// TwinCAT 3 PLC project PLCStudent
// ProgramVersion: 3.1.4022.3
// libraries:
//   Tc2_Standard, * (Beckhoff Automation GmbH)
//   Tc2_System, * (Beckhoff Automation GmbH)
//   Tc3_Module, * (Beckhoff Automation GmbH)
// project tree:
//   GVLs/ GVL.TcGVL
//   / PlcTask.TcTTO (not stored)
//   POUs/ MAIN.TcPOU, Wash.TcPOU
// (motion and I/O tree: see PLC project plcsim)
// real-time tasks:
//   TASK PlcTask: cycle T#80ms, priority 1, ADS port 350
//   TASK PlcTask1: cycle T#10ms, priority 20, ADS port 351
// variable links:
//   PLCSim/PLCSim Instance <-> PLCStudent/PLCStudent Instance
//     PlcTask Inputs/GVL.ixBack <-> PlcTask Outputs/GVL.qxBack
//     PlcTask Inputs/GVL.ixDispBit1 <-> PlcTask Outputs/GVL.qxDispBit1
//     PlcTask Inputs/GVL.ixDispBit2 <-> PlcTask Outputs/GVL.qxDispBit2
//     PlcTask Inputs/GVL.ixDrain <-> PlcTask Outputs/GVL.qxDrain
//     PlcTask Inputs/GVL.ixFill <-> PlcTask Outputs/GVL.qxFill
//     PlcTask Inputs/GVL.ixForw <-> PlcTask Outputs/GVL.qxForw
//     PlcTask Inputs/GVL.ixHeating <-> PlcTask Outputs/GVL.qxHeatingON
//     PlcTask Inputs/GVL.ixPulseTwo <-> PlcTask Outputs/GVL.qxPulseTwo
//     PlcTask Inputs/GVL.ixSpin <-> PlcTask Outputs/GVL.qxSpin
//     PlcTask Outputs/GVL.qwCurTemp <-> PlcTask Inputs/GVL.iwCurrentTemp
//     PlcTask Outputs/GVL.qwSetTem <-> PlcTask Inputs/GVL.iwSetTemp
//     PlcTask Outputs/GVL.qxLevel1 <-> PlcTask Inputs/GVL.ixLevel1
//     PlcTask Outputs/GVL.qxLevel2 <-> PlcTask Inputs/GVL.ixLevel2
//     PlcTask Outputs/GVL.qxLevel3 <-> PlcTask Inputs/GVL.ixLevel3
//     PlcTask Outputs/GVL.qxNotEmpty <-> PlcTask Inputs/GVL.ixNotEmpty
//     PlcTask Outputs/GVL.qxPulseOne <-> PlcTask Inputs/GVL.ixPulseOne
//     PlcTask Outputs/GVL.qxSetLevel <-> PlcTask Inputs/GVL.ixSetLevel
//     PlcTask Outputs/GVL.qxStart <-> PlcTask Inputs/GVL.ixStart
//     PlcTask Outputs/GVL.qxTempOk <-> PlcTask Inputs/GVL.ixTempOk

// ---- GVLs/GVL.TcGVL
{attribute 'qualified_only'}
VAR_GLOBAL
	ixPulseOne		AT %I*:	BOOL; 		(* PULS button *)
	ixStart			AT %I*:	BOOL; 		(* START switch *)
	ixSetLevel		AT %I*:	BOOL; 		(* NIVÅ switch *)
	ixLevel3		AT %I*:	BOOL; 		(* Sensor for level 3 *)
	ixLevel2		AT %I*:	BOOL; 		(* Sensor for level 2 *)
	ixLevel1		AT %I*:	BOOL; 		(* Sensor for level 1 *)
	ixNotEmpty		AT %I*:	BOOL; 		(* Sensor for not empty *)
	ixTempOk		AT %I*:	BOOL; 		(* Temp sensor *)
	iwSetTemp		AT %I*: INT;		(* Temparature set on the dail in HMI*)
	iwCurrentTemp	AT %I*: INT;		(* Current Temparture of the washing machine*)
	
	qxPulseTwo		AT %Q*:	BOOL; 		(* PULS button *)
	qxForw			AT %Q*:	BOOL; 		(* Washer cylinder forward *)
	qxBack			AT %Q*:	BOOL; 		(* Washer cylinder back *)
	qxSpin			AT %Q*:	BOOL; 		(* Washer cylinder spin *)
	qxFill			AT %Q*:	BOOL; 		(* Fill water *)
	qxDrain			AT %Q*:	BOOL; 		(* Drain water *)
	qxDispBit1		AT %Q*:	BOOL; 		(* Display bit 1 *)
	qxDispBit2		AT %Q*:	BOOL; 		(* Display bit 2 *)
	qxHeatingON		AT %Q*: BOOL;		(* Heater ON *)
END_VAR

// ---- POUs/MAIN.TcPOU
PROGRAM MAIN
VAR
END_VAR

Wash();

END_PROGRAM

// ---- POUs/Wash.TcPOU
PROGRAM Wash
VAR
	Blink_Timer: TP;
	Stop_Timer: TON;
	Memorize: BOOL;
END_VAR

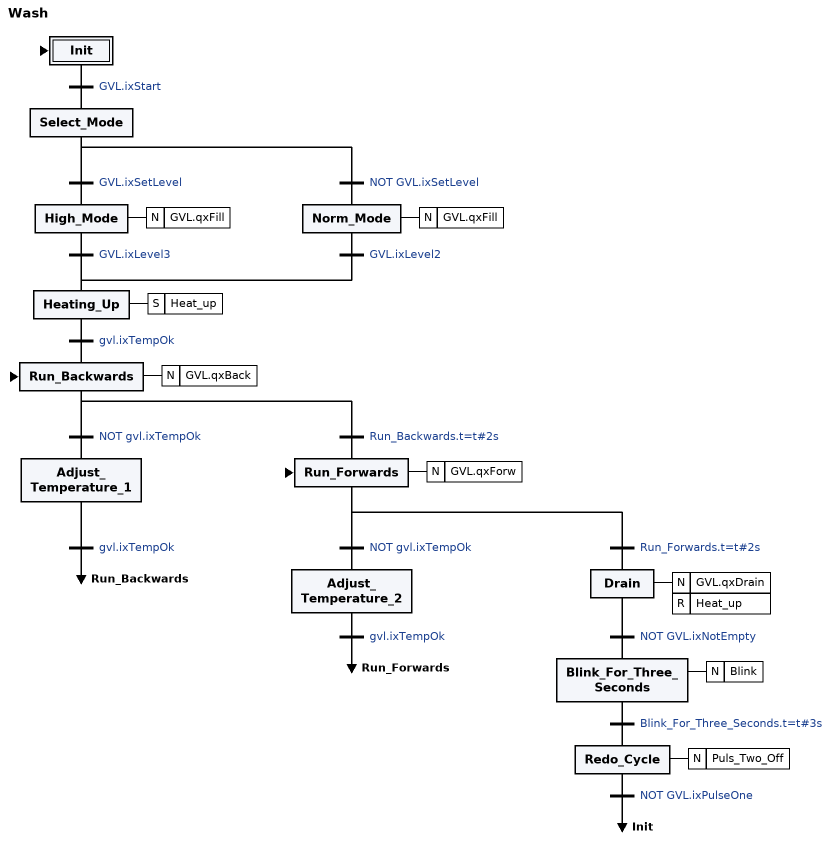
INITIAL_STEP Init:
END_STEP
TRANSITION FROM Init TO Select_Mode
    := GVL.ixStart;
END_TRANSITION
STEP Select_Mode:
END_STEP
TRANSITION FROM Select_Mode TO High_Mode
    := GVL.ixSetLevel;
END_TRANSITION
STEP High_Mode:
    GVL.qxFill(N);
END_STEP
TRANSITION FROM High_Mode TO Heating_Up
    := GVL.ixLevel3;
END_TRANSITION
TRANSITION FROM Select_Mode TO Norm_Mode
    := NOT GVL.ixSetLevel;
END_TRANSITION
STEP Norm_Mode:
    GVL.qxFill(N);
END_STEP
TRANSITION FROM Norm_Mode TO Heating_Up
    := GVL.ixLevel2;
END_TRANSITION
STEP Heating_Up:
    Heat_up(S);
END_STEP
TRANSITION FROM Heating_Up TO Run_Backwards
    := gvl.ixTempOk;
END_TRANSITION
STEP Run_Backwards:
    GVL.qxBack(N);
END_STEP
TRANSITION FROM Run_Backwards TO Adjust_Temperature_1
    := NOT gvl.ixTempOk;
END_TRANSITION
STEP Adjust_Temperature_1:
END_STEP
TRANSITION FROM Adjust_Temperature_1 TO Run_Backwards
    := gvl.ixTempOk;
END_TRANSITION
TRANSITION FROM Run_Backwards TO Run_Forwards
    := Run_Backwards.t=t#2s;
END_TRANSITION
STEP Run_Forwards:
    GVL.qxForw(N);
END_STEP
TRANSITION FROM Run_Forwards TO Adjust_Temperature_2
    := NOT gvl.ixTempOk;
END_TRANSITION
STEP Adjust_Temperature_2:
END_STEP
TRANSITION FROM Adjust_Temperature_2 TO Run_Forwards
    := gvl.ixTempOk;
END_TRANSITION
TRANSITION FROM Run_Forwards TO Drain
    := Run_Forwards.t=t#2s;
END_TRANSITION
STEP Drain:
    GVL.qxDrain(N);
    Heat_up(R);
END_STEP
TRANSITION FROM Drain TO Blink_For_Three_Seconds
    := NOT GVL.ixNotEmpty;
END_TRANSITION
STEP Blink_For_Three_Seconds:
    Blink(N);
END_STEP
TRANSITION FROM Blink_For_Three_Seconds TO Redo_Cycle
    := Blink_For_Three_Seconds.t=t#3s;
END_TRANSITION
STEP Redo_Cycle:
    Puls_Two_Off(N);
END_STEP
TRANSITION FROM Redo_Cycle TO Init
    := NOT GVL.ixPulseOne;
END_TRANSITION

ACTION Blink:
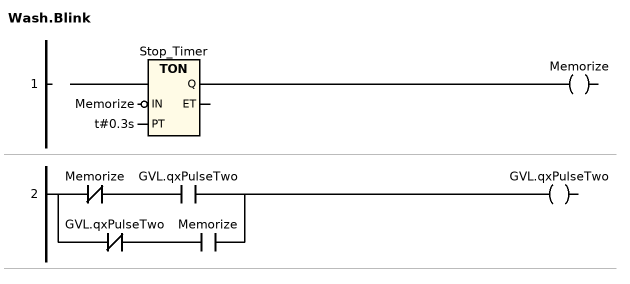
// NETWORK 1
Stop_Timer(IN := NOT Memorize, PT := t#0.3s); // TON
Memorize := Stop_Timer.Q;

// NETWORK 2
GVL.qxPulseTwo := NOT Memorize AND GVL.qxPulseTwo OR NOT GVL.qxPulseTwo AND Memorize;
END_ACTION

ACTION Heat_up:
IF gvl.iwCurrentTemp<=gvl.iwSetTemp THEN
	GVL.qxHeatingON := TRUE;
	
ELSE
	GVL.qxHeatingON := FALSE;
END_IF
END_ACTION

ACTION Puls_Two_Off:
gvl.qxPulseTwo:=FALSE;
END_ACTION

ACTION Reheat:

END_ACTION

END_PROGRAM
